{attribute addProperty BoxType "KL2642-0050"}
{attribute addProperty Id "State_RelayAT %I*BOOL000OutputAT %Q*BOOL000"}
{attribute addProperty CRC "1022788430"}
{attribute addProperty SizeInBites "0"}
{attribute addProperty SizeInBytes "0"}
TYPE Channel_3CF6834E :
STRUCT
	{attribute addProperty Name "State_Relay"}
	State_Relay AT %I* : BOOL;
	{attribute addProperty Name "Output"}
	Output AT %Q* : BOOL;
END_STRUCT
END_TYPE

(* stored: Version 1.2.0.0, ProductVersion 3.1.4024.9
   DUT Channel_3CF6834E: Id {9879d2ae-268d-4dd1-a815-896ec3cf614e} *)
